{attribute addProperty BoxType "EL6201-0000-0017"}
{attribute addProperty Id "Slave_5A_DO0BIT10.12533Slave_5A_DO1BIT10.12534Slave_5A_DO2BIT10.12535Slave_5A_DO3BIT10.12536Slave_5B_DO0BIT10.12537Slave_5B_DO1BIT10.12538Slave_5B_DO2BIT10.12539Slave_5B_DO3BIT10.12540"}
{attribute addProperty CRC "1344951697"}
{attribute addProperty SizeInBites "8"}
{attribute addProperty SizeInBytes "1"}
TYPE Slave_5_Outputs_502A5591 :
STRUCT
	{attribute addProperty Name "Slave_5A_DO0"}
	Slave_5A_DO0 : BIT;
	{attribute addProperty Name "Slave_5A_DO1"}
	Slave_5A_DO1 : BIT;
	{attribute addProperty Name "Slave_5A_DO2"}
	Slave_5A_DO2 : BIT;
	{attribute addProperty Name "Slave_5A_DO3"}
	Slave_5A_DO3 : BIT;
	{attribute addProperty Name "Slave_5B_DO0"}
	Slave_5B_DO0 : BIT;
	{attribute addProperty Name "Slave_5B_DO1"}
	Slave_5B_DO1 : BIT;
	{attribute addProperty Name "Slave_5B_DO2"}
	Slave_5B_DO2 : BIT;
	{attribute addProperty Name "Slave_5B_DO3"}
	Slave_5B_DO3 : BIT;
END_STRUCT
END_TYPE

(* stored: Version 1.2.0.0, ProductVersion 3.1.4024.9
   DUT Slave_5_Outputs_502A5591: Id {5896ede2-386b-491c-9e7c-83c79930ddd5} *)
